METHOD Completing : BOOL
VAR_INPUT
    SequenceState : REFERENCE TO UDINT;
END_VAR
Completing := TRUE;
END_METHOD

METHOD Execute : BOOL
VAR_INPUT
    SequenceState : REFERENCE TO UDINT;
END_VAR
Execute := TRUE;
END_METHOD

METHOD Held : BOOL
VAR_INPUT
    SequenceState : REFERENCE TO UDINT;
END_VAR
Held := TRUE;
END_METHOD

METHOD Holding : BOOL
VAR_INPUT
    SequenceState : REFERENCE TO UDINT;
END_VAR
Holding := TRUE;
END_METHOD

METHOD Idle : BOOL
VAR_INPUT
    SequenceState : REFERENCE TO UDINT;
END_VAR
Idle := TRUE;
END_METHOD

METHOD Resetting : BOOL
VAR_INPUT
    SequenceState : REFERENCE TO UDINT;
END_VAR
Resetting := TRUE;
END_METHOD

METHOD Starting : BOOL
VAR_INPUT
    SequenceState : REFERENCE TO UDINT;
END_VAR
Starting := TRUE;
END_METHOD

METHOD Stopped : BOOL
VAR_INPUT
    SequenceState : REFERENCE TO UDINT;
END_VAR
Stopped := TRUE;
END_METHOD

METHOD Stopping : BOOL
VAR_INPUT
    SequenceState : REFERENCE TO UDINT;
END_VAR
Stopping := TRUE;
END_METHOD

METHOD Suspended : BOOL
VAR_INPUT
    SequenceState : REFERENCE TO UDINT;
END_VAR
Suspended := TRUE;
END_METHOD

METHOD Suspending : BOOL
VAR_INPUT
    SequenceState : REFERENCE TO UDINT;
END_VAR
Suspending := TRUE;
END_METHOD

METHOD Unholding : BOOL
VAR_INPUT
    SequenceState : REFERENCE TO UDINT;
END_VAR
Unholding := TRUE;
END_METHOD

METHOD Unsuspending : BOOL
VAR_INPUT
    SequenceState : REFERENCE TO UDINT;
END_VAR
Unsuspending := TRUE;
END_METHOD

(* This Module will be done initialize when ModuleInitialized := TRUE;, subequently all subitems will be called to be initialized *)
METHOD Initializing
END_METHOD

METHOD OnCyclicCall
END_METHOD

PROPERTY Statemachine : I_Statemachine
GET
Statemachine := _Statemachine;
END_GET
END_PROPERTY

END_FUNCTION_BLOCK

// Statemachine/PackML/PackMLStatemachine
FUNCTION_BLOCK PackMLStatemachine EXTENDS CyclicComponent IMPLEMENTS I_StateMachine
VAR
	StateList	   : StateList<17>;
	StateMachine   : FB_PMLStateMachine;
	StateCommand   : E_PMLCommand;
	_CurrentState  : E_PMLState;
	ModeController : PackMLModeControl := (StateMachine := THIS^);
END_VAR

PROPERTY Mode : I_Mode
GET
Mode := ModeController;
END_GET
SET
// Fix defined in PackML
END_SET
END_PROPERTY

METHOD PROTECTED CallState : BOOL
VAR_INPUT
	StateIndex : E_PMLState;
END_VAR

VAR
	State : I_State;
	i	  : DINT;
END_VAR
State := StateList.GetStateAtIndex(StateIndex);
IF State <> 0 THEN
	CallState := State.Executing();
ELSE
	CallState := TRUE;
END_IF

FOR i := 0 TO StateList.NumberOfStates DO
	State := StateList.GetStateAtIndex(i);
	IF State <> 0 AND i <> StateIndex THEN
		State.Inactive();
	END_IF
END_FOR
END_METHOD

METHOD ChangeState
VAR_INPUT
	StateCommand : DINT;
END_VAR
IF StateCommand <= 0 OR StateCommand > 17 THEN
	Trace.LogMessage('PackML Statemachine ChangeState()', 'StateId is not a PackML State');
END_IF

{warning disable C0196}
THIS^.StateCommand := StateCommand;
END_METHOD

{attribute 'monitoring' := 'call'}
PROPERTY CurrentState : DINT
GET
CurrentState := _CurrentState;
END_GET
END_PROPERTY

PROPERTY States : I_StateList
GET
States := StateList;
END_GET
END_PROPERTY

METHOD CyclicLogic
VAR_INST
	ClearingTon : TON;
END_VAR
IF StateList.NumberOfStates = 0 THEN
	RETURN;
END_IF

ModeController.CyclicLogic();
IF _CurrentState = E_PMLState.Undefined AND Mode.CurrentMode <> 0 THEN
	StateCommand := E_PMLCommand.Abort;
END_IF

StateMachine(eMode			  := TO_DINT(Mode.CurrentMode),
			 eCommand		  := StateCommand,
			 stSubUnitInfoRef :=,
			 stOptions		  :=,
			 eState			  => _CurrentState,
			 sState			  =>,
			 bError			  =>,
			 nErrorID		  =>);

CASE _CurrentState OF
	E_PMLState.Undefined:
		CallState(_CurrentState);

	E_PMLState.Clearing:
		ClearingTon(IN := TRUE, PT := CoreParameter.ClearingTimeout);
		IF CallState(_CurrentState) THEN
			ClearingTon(IN := FALSE);
			StateMachine.M_StateComplete();
		END_IF

		IF ClearingTon.Q THEN
			ClearingTon(IN := FALSE);
			Trace.LogMessage('Clearing Timeout exeeded!', 'CoreParameter.ClearingTimeout');
			StateCommand := E_PMLCommand.Abort;
		END_IF

	E_PMLState.Stopped:
		CallState(_CurrentState);

	E_PMLState.Starting:
		IF CallState(_CurrentState) THEN
			StateMachine.M_StateComplete();
		END_IF

	E_PMLState.Idle:
		CallState(_CurrentState);

	E_PMLState.Suspended:
		CallState(_CurrentState);

	E_PMLState.Execute:
		CallState(_CurrentState);

	E_PMLState.Stopping:
		IF CallState(_CurrentState) THEN
			StateMachine.M_StateComplete();
		END_IF

	E_PMLState.Aborting:
		IF CallState(_CurrentState) THEN
			StateMachine.M_StateComplete();
		END_IF

	E_PMLState.Aborted:
		CallState(_CurrentState);

	E_PMLState.Holding:
		IF CallState(_CurrentState) THEN
			StateMachine.M_StateComplete();
		END_IF

	E_PMLState.Held:
		CallState(_CurrentState);

	E_PMLState.Unholding:
		IF CallState(_CurrentState) THEN
			StateMachine.M_StateComplete();
		END_IF

	E_PMLState.Suspending:
		IF CallState(_CurrentState) THEN
			StateMachine.M_StateComplete();
		END_IF

	E_PMLState.Unsuspending:
		IF CallState(_CurrentState) THEN
			StateMachine.M_StateComplete();
		END_IF

	E_PMLState.Resetting:
		IF CallState(_CurrentState) THEN
			StateMachine.M_StateComplete();
		END_IF

	E_PMLState.Completing:
		IF CallState(_CurrentState) THEN
			StateMachine.M_StateComplete();
		END_IF

	E_PMLState.Completed:
		CallState(_CurrentState);
END_CASE
END_METHOD

END_FUNCTION_BLOCK

// Project Information/F_GetCompany
// This function has been automatically generated from the project information.
{attribute 'signature_flag' := '1073741824'}
{attribute 'TcGenerated'}
{attribute 'no-analysis'}
FUNCTION F_GetCompany : WSTRING
VAR_INPUT
	
END_VAR

F_GetCompany := "Beckhoff Automation LLC";

END_FUNCTION

// Project Information/F_GetTitle
// This function has been automatically generated from the project information.
{attribute 'signature_flag' := '1073741824'}
{attribute 'TcGenerated'}
{attribute 'no-analysis'}
FUNCTION F_GetTitle : WSTRING
VAR_INPUT
	
END_VAR

F_GetTitle := "Core";

END_FUNCTION

// Project Information/F_GetVersion
// This function has been automatically generated from the project information.
{attribute 'signature_flag' := '1073741824'}
{attribute 'TcGenerated'}
{attribute 'no-analysis'}
FUNCTION F_GetVersion : ST_LibVersion
VAR_INPUT
	
END_VAR

F_GetVersion.iMajor := 1;
F_GetVersion.iMinor := 2;
F_GetVersion.iBuild := 0;
F_GetVersion.iRevision := 0;
F_GetVersion.sVersion := '1.2.0';
F_GetVersion.nFlags := 0;

END_FUNCTION

// Statemachine/Generic/NextMinorStep
FUNCTION NextMinorStep : UDINT
VAR_IN_OUT
	StateVar : UDINT;
END_VAR

NextMinorStep := StateVar := StateVar + 1;

END_FUNCTION

// Statemachine/Generic/NextStep
FUNCTION NextStep : UDINT
VAR_IN_OUT
	StateVar : UDINT;
END_VAR

NextStep := StateVar := ((StateVar / 10) * 10) + 10;

END_FUNCTION

// Statemachine/Generic/Statemachine_HMI
FUNCTION_BLOCK Statemachine_HMI EXTENDS HmiFunction
VAR
	Statemachine : I_Statemachine;
	{ attribute 'TcHmiSymbol.AddSymbol' }
	{ attribute 'TcHmiSymbol.AddSymbol.UserGroups' := '__SystemAdministrators,Admin' }
	Statemachine_HMI : ST_Statemachine_HMI;
END_VAR

METHOD CyclicLogic
VAR_INST
	LastModeChangeCommand  : DINT;
	LastStateChangeCommand : DINT;
END_VAR
Statemachine_HMI.Name		  := Statemachine.Name;
Statemachine_HMI.CurrentState := Statemachine.CurrentState;
Statemachine_HMI.CurrentMode  := Statemachine.Mode.CurrentMode;
Statemachine_HMI.HmiEnabled	  := Enabled;
IF Enabled THEN
	IF Statemachine_HMI.ModeChangeCommand <> 0 THEN
		Statemachine.Mode.ChangeMode(Statemachine_HMI.ModeChangeCommand);
		LastModeChangeCommand			   := Statemachine_HMI.ModeChangeCommand;
		Statemachine_HMI.ModeChangeCommand := 0;
	END_IF

	{warning disable C0196}
	IF Statemachine_HMI.StateChangeCommand <> 0 THEN
		Statemachine.ChangeState(TO_UDINT(Statemachine_HMI.StateChangeCommand));
		{warning disable C0195}
		LastStateChangeCommand				:= Statemachine_HMI.StateChangeCommand;
		Statemachine_HMI.StateChangeCommand := 0;
	END_IF
ELSE
	Statemachine_HMI.StateChangeCommand := 0;
	Statemachine_HMI.ModeChangeCommand	:= 0;
END_IF
END_METHOD

(*FB_Init is always available implicitly and it is used primarily for initialization.
The return value is not evaluated. For a specific influence, you can also declare the
methods explicitly and provide additional code there with the standard initialization
code. You can evaluate the return value.*)
METHOD FB_Init : BOOL
VAR_INPUT
	(* TRUE: the retain variables are initialized (reset warm / reset cold)*)
	bInitRetains : BOOL;

	(* TRUE: the instance will be copied to the copy code afterward (online change)   *)
	bInCopyCode	 : BOOL;
	Name		 : T_MaxString;
	Statemachine : I_Statemachine;
END_VAR
THIS^.Statemachine := Statemachine;
ControlType		   := 'Statemachine';
LinkObject		   := 'Statemachine_HMI';
END_METHOD

END_FUNCTION_BLOCK

// Statemachine/PackML/NextAvailablePackMLCommands
FUNCTION_BLOCK NextAvailablePackMLCommands
VAR
	NextAvailableCommands : ARRAY[0..MAX_AVAILABLE_COMMANDS] OF E_PMLCommand;
	i					  : UDINT;
END_VAR

VAR CONSTANT
	MAX_AVAILABLE_COMMANDS : UDINT := 9;
END_VAR

METHOD PUBLIC GetCommands : ARRAY[0..MAX_AVAILABLE_COMMANDS] OF E_PMLCommand
VAR_INPUT
	CurrentMode	 : DINT(0..31);
	CurrentState : E_PMLState;
END_VAR

VAR
	ModeConfiguration : Tc3_PackML_V3.ST_PMLUnitModeConfiguration;
END_VAR
FOR i := 1 TO MAX_AVAILABLE_COMMANDS DO
	NextAvailableCommands[i] := E_PMLCommand.Undefined;
END_FOR

i				  := 0;
ModeConfiguration := Tc3_PackML_V3.GlobalVariables.stPMLUnitModeConfiguration[CurrentMode];
// Generate next possible Commands
CASE CurrentState OF
	E_PMLState.Undefined:
		;

	E_PMLState.Aborting:
		;

	E_PMLState.Aborted:
		NextAvailableCommands[i] := E_PMLCommand.Clear;

	E_PMLState.Clearing:
		;

	E_PMLState.Stopping:
		NextAvailableCommands[i] := E_PMLCommand.Abort;

	E_PMLState.Stopped:
		NextAvailableCommands[i] := E_PMLCommand.Abort;
		i						 := i + 1;
		IF NOT ModeConfiguration.aStateDisabled[E_PMLState.Resetting] AND NOT ModeConfiguration.aStateDisabled[E_PMLState.Idle] THEN
			NextAvailableCommands[i] := E_PMLCommand.Reset;
		ELSE
			NextAvailableCommands[i] := E_PMLCommand.Start;
		END_IF

	E_PMLState.Resetting:
		NextAvailableCommands[i] := E_PMLCommand.Abort;
		i						 := i + 1;
		NextAvailableCommands[i] := E_PMLCommand.Stop;

	E_PMLState.Idle:
		NextAvailableCommands[i] := E_PMLCommand.Abort;
		i						 := i + 1;
		NextAvailableCommands[i] := E_PMLCommand.Stop;
		i						 := i + 1;
		NextAvailableCommands[i] := E_PMLCommand.Start;

	E_PMLState.Starting:
		NextAvailableCommands[i] := E_PMLCommand.Abort;
		i						 := i + 1;
		NextAvailableCommands[i] := E_PMLCommand.Stop;

	E_PMLState.Execute:
		NextAvailableCommands[i] := E_PMLCommand.Abort;
		i						 := i + 1;
		NextAvailableCommands[i] := E_PMLCommand.Stop;
		i						 := i + 1;
		IF (NOT ModeConfiguration.aStateDisabled[E_PMLState.Held] AND NOT ModeConfiguration.aStateDisabled[E_PMLState.Holding]) OR (NOT ModeConfiguration.aStateDisabled[E_PMLState.Held] AND NOT ModeConfiguration.aStateDisabled[E_PMLState.Unholding]) THEN
			NextAvailableCommands[i] := E_PMLCommand.Hold;
			i						 := i + 1;
		END_IF

		IF (NOT ModeConfiguration.aStateDisabled[E_PMLState.Suspended] AND NOT ModeConfiguration.aStateDisabled[E_PMLState.Suspending]) OR (NOT ModeConfiguration.aStateDisabled[E_PMLState.Suspended] AND NOT ModeConfiguration.aStateDisabled[E_PMLState.Unsuspending]) THEN
			NextAvailableCommands[i] := E_PMLCommand.Suspend;
			i						 := i + 1;
		END_IF

		IF NOT ModeConfiguration.aStateDisabled[E_PMLState.Completed] AND NOT ModeConfiguration.aStateDisabled[E_PMLState.Completing] THEN
			NextAvailableCommands[i] := E_PMLCommand.Complete;
			i						 := i + 1;
		ELSIF NOT ModeConfiguration.aStateDisabled[E_PMLState.Resetting] THEN
			NextAvailableCommands[i] := E_PMLCommand.Reset;
			i						 := i + 1;
		END_IF

	E_PMLState.Completing:
		NextAvailableCommands[i] := E_PMLCommand.Abort;
		i						 := i + 1;
		NextAvailableCommands[i] := E_PMLCommand.Stop;

	E_PMLState.Completed:
		NextAvailableCommands[i] := E_PMLCommand.Abort;
		i						 := i + 1;
		NextAvailableCommands[i] := E_PMLCommand.Stop;
		i						 := i + 1;
		IF NOT ModeConfiguration.aStateDisabled[E_PMLState.Resetting] AND NOT ModeConfiguration.aStateDisabled[E_PMLState.Idle] THEN
			NextAvailableCommands[i] := E_PMLCommand.Reset;
		ELSE
			NextAvailableCommands[i] := E_PMLCommand.Start;
		END_IF

	E_PMLState.Holding:
		NextAvailableCommands[i] := E_PMLCommand.Abort;
		i						 := i + 1;
		NextAvailableCommands[i] := E_PMLCommand.Stop;

	E_PMLState.Held:
		NextAvailableCommands[i] := E_PMLCommand.Abort;
		i						 := i + 1;
		NextAvailableCommands[i] := E_PMLCommand.Stop;
		i						 := i + 1;
		NextAvailableCommands[i] := E_PMLCommand.Unhold;

	E_PMLState.Unholding:
		NextAvailableCommands[i] := E_PMLCommand.Abort;
		i						 := i + 1;
		NextAvailableCommands[i] := E_PMLCommand.Stop;

	E_PMLState.Suspending:
		NextAvailableCommands[i] := E_PMLCommand.Abort;
		i						 := i + 1;
		NextAvailableCommands[i] := E_PMLCommand.Stop;

	E_PMLState.Suspended:
		NextAvailableCommands[i] := E_PMLCommand.Abort;
		i						 := i + 1;
		NextAvailableCommands[i] := E_PMLCommand.Stop;
		i						 := i + 1;
		NextAvailableCommands[i] := E_PMLCommand.Unsuspend;

	E_PMLState.Unsuspending:
		NextAvailableCommands[i] := E_PMLCommand.Abort;
		i						 := i + 1;
		NextAvailableCommands[i] := E_PMLCommand.Stop;
END_CASE

GetCommands := NextAvailableCommands;
END_METHOD

END_FUNCTION_BLOCK

// Statemachine/PackML/PackMLStatemachine_HMI
FUNCTION_BLOCK PackMLStatemachine_HMI EXTENDS HmiFunction
VAR
	Statemachine				: I_Statemachine;
	NextAvailablePackMLCommands : NextAvailablePackMLCommands;
	{ attribute 'TcHmiSymbol.AddSymbol' }
	{ attribute 'TcHmiSymbol.AddSymbol.UserGroups' := '__SystemAdministrators,Admin' }
	Statemachine_HMI : ST_PackMLStatemachine_HMI;
END_VAR

METHOD CyclicLogic
VAR_INST
	LastModeChangeCommand  : DINT;
	LastStateChangeCommand : UDINT;
END_VAR
{warning disable C0196}
Statemachine_HMI.CurrentState := Statemachine.CurrentState;
Statemachine_HMI.CurrentMode  := Statemachine.Mode.CurrentMode;
Statemachine_HMI.Name		  := Statemachine.Name;
Statemachine_HMI.HmiEnabled	  := Enabled;
IF Enabled THEN
	IF Statemachine_HMI.ModeCommand <> 0 THEN
		Statemachine.Mode.ChangeMode(Statemachine_HMI.ModeCommand);
		LastModeChangeCommand		 := Statemachine_HMI.ModeCommand;
		Statemachine_HMI.ModeCommand := 0;
	END_IF

	{warning disable C0196}
	IF Statemachine_HMI.StateCommand <> 0 THEN
		Statemachine.ChangeState(TO_UDINT(Statemachine_HMI.StateCommand));
		{warning disable C0195}
		LastStateChangeCommand		  := Statemachine_HMI.StateCommand;
		Statemachine_HMI.StateCommand := 0;
	END_IF
ELSE
	Statemachine_HMI.StateCommand := 0;
	Statemachine_HMI.ModeCommand  := 0;
END_IF

Statemachine_HMI.NextAvailableCommands := NextAvailablePackMLCommands.GetCommands(Statemachine_HMI.CurrentMode, Statemachine_HMI.CurrentState);
END_METHOD

(*FB_Init is always available implicitly and it is used primarily for initialization.
The return value is not evaluated. For a specific influence, you can also declare the
methods explicitly and provide additional code there with the standard initialization
code. You can evaluate the return value.*)
METHOD FB_Init : BOOL
VAR_INPUT
	(* TRUE: the retain variables are initialized (reset warm / reset cold)*)
	bInitRetains : BOOL;

	(* TRUE: the instance will be copied to the copy code afterward (online change)   *)
	bInCopyCode	 : BOOL;
	Name		 : T_MaxString;
	Statemachine : I_Statemachine;
END_VAR
THIS^.Statemachine := Statemachine;
ControlType		   := 'PackMLStatemachine';
LinkObject		   := 'Statemachine_HMI';
END_METHOD

END_FUNCTION_BLOCK

// Visitors/Enable/CheckComponentsEnabledVisitor
FUNCTION_BLOCK CheckComponentsEnabledVisitor IMPLEMENTS I_ComponentVisitor
VAR
	Enablable : I_Enablable;
	_Enabled  : BOOL;
END_VAR

METHOD Check
VAR_INPUT
	Components : I_ComponentCollection;
END_VAR
_Enabled := TRUE;
Components.Accept(THIS^);
END_METHOD

{attribute 'monitoring' := 'call'}
PROPERTY Enabled : BOOL
GET
Enabled := _Enabled;
END_GET
END_PROPERTY

METHOD VisitComponent
VAR_INPUT
	Component : I_Component;
END_VAR
IF __QUERYINTERFACE(Component, Enablable) THEN
	IF NOT Enablable.Enabled THEN
		_Enabled := FALSE;
	END_IF
END_IF
END_METHOD

END_FUNCTION_BLOCK

// Visitors/Enable/DisableAllComponentsVisitor
FUNCTION_BLOCK DisableAllComponentsVisitor IMPLEMENTS I_ComponentVisitor
VAR
	Enablable : I_Enablable;
	_Enabled  : BOOL;
END_VAR

METHOD Disable
VAR_INPUT
	Components : I_ComponentCollection;
END_VAR
_Enabled := FALSE;
Components.Accept(THIS^);
END_METHOD

{attribute 'monitoring' := 'call'}
PROPERTY Enabled : BOOL
GET
Enabled := _Enabled;
END_GET
END_PROPERTY

METHOD VisitComponent
VAR_INPUT
	Component : I_Component;
END_VAR
IF __QUERYINTERFACE(Component, Enablable) THEN
	Enablable.Disable();
	IF Enablable.Enabled THEN
		_Enabled := TRUE;
	END_IF
END_IF
END_METHOD

END_FUNCTION_BLOCK

// Visitors/Enable/EnableAllComponentsVisitor
FUNCTION_BLOCK EnableAllComponentsVisitor IMPLEMENTS I_ComponentVisitor
VAR
	Enablable	   : I_Enablable;
	_Enabled	   : BOOL;
	ErrorComponent : I_Component;
END_VAR

METHOD Enable
VAR_INPUT
	Components : I_ComponentCollection;
END_VAR
_Enabled := TRUE;
Components.Accept(THIS^);
END_METHOD

{attribute 'monitoring' := 'call'}
PROPERTY Enabled : BOOL
GET
Enabled := _Enabled;
END_GET
END_PROPERTY

METHOD VisitComponent
VAR_INPUT
	Component : I_Component;
END_VAR
IF __QUERYINTERFACE(Component, Enablable) THEN
	Enablable.Enable();
	IF NOT Enablable.Enabled THEN
		ErrorComponent := Component;
		_Enabled	   := FALSE;
	END_IF
END_IF
END_METHOD

END_FUNCTION_BLOCK

// Visitors/Events/GetActiveEventSeverityVisitor
FUNCTION_BLOCK GetActiveEventSeverityVisitor IMPLEMENTS I_ModuleVisitor, I_ComponentVisitor
VAR
	EntryModule			 : I_Module;
	HighestEventSeverity : TcEventSeverity;
	TcEventClass		 : I_EventClassTcEvents;
END_VAR

PROPERTY ActiveEventSeverity : TcEventSeverity
GET
HighestEventSeverity := Global.TcEventSeverity.Verbose;
EntryModule.Accept(THIS^);
ActiveEventSeverity := HighestEventSeverity;
END_GET
END_PROPERTY

(*FB_Init is always available implicitly and it is used primarily for initialization.
The return value is not evaluated. For a specific influence, you can also declare the
methods explicitly and provide additional code there with the standard initialization
code. You can evaluate the return value.*)
METHOD FB_Init : BOOL
VAR_INPUT
	(* TRUE: the retain variables are initialized (reset warm / reset cold)*)
	bInitRetains : BOOL;

	(* TRUE: the instance will be copied to the copy code afterward (online change)   *)
	bInCopyCode : BOOL;
	EntryModule : I_Module;
END_VAR
THIS^.EntryModule := EntryModule;
END_METHOD

METHOD VisitComponent
VAR_INPUT
	Component : I_Component;
END_VAR

VAR
	Severity : TcEventSeverity;
END_VAR
IF __QUERYINTERFACE(Component, TcEventClass) THEN
	Severity := TcEventClass.GetHighestActiveEventSeverity();
	IF Severity > HighestEventSeverity THEN
		HighestEventSeverity := Severity;
	END_IF
END_IF
END_METHOD

METHOD VisitModule
VAR_INPUT
	Module : I_Module;
END_VAR

VAR
	Severity : TcEventSeverity;
END_VAR
Module.Components.Accept(THIS^);
Module.Modules.Accept(THIS^);
IF __QUERYINTERFACE(Module, TcEventClass) THEN
	Severity := TcEventClass.GetHighestActiveEventSeverity();
	IF Severity > HighestEventSeverity THEN
		HighestEventSeverity := Severity;
	END_IF
END_IF
END_METHOD

END_FUNCTION_BLOCK

// Visitors/HMI/GetSystemTreeJsonHmiVisitor
FUNCTION_BLOCK GetSystemTreeJsonHmiVisitor
VAR_GENERIC CONSTANT
	TreeMax : UDINT := 10000;
END_VAR IMPLEMENTS I_ModuleVisitor, I_ComponentVisitor
VAR
	{ attribute 'TcHmiSymbol.AddSymbol' }
	{ attribute 'TcHmiSymbol.AddSymbol.UserGroups' := '__SystemAdministrators,Admin' }
	SystemHmiTree : STRING(TreeMax);
	{attribute 'hide'}
	Module : I_Module;
	{attribute 'hide'}
	HmiFunction : I_HmiFunction;
	{attribute 'hide'}
	Json : FB_JsonSaxWriter;
	{attribute 'hide'}
	Entry	 : T_MaxString;
	LinkRoot : STRING;
END_VAR

METHOD PRIVATE Clear
VAR_INPUT
END_VAR
MEMSET(ADR(SystemHmiTree), 0, SIZEOF(SystemHmiTree));
Json.ResetDocument();
END_METHOD

//FB_Init is always available implicitly and it is used primarily for initialization.

//The return value is not evaluated. For a specific influence, you can also declare the

//methods explicitly and provide additional code there with the standard initialization

//code. You can evaluate the return value.
METHOD FB_Init : BOOL
VAR_INPUT
	bInitRetains : BOOL; // TRUE: the retain variables are initialized (reset warm / reset cold)
	bInCopyCode	 : BOOL; // TRUE: the instance will be copied to the copy code afterward (online change)   
	LinkRoot	 : STRING;
END_VAR
THIS^.LinkRoot := LinkRoot;
END_METHOD

METHOD GetTree
VAR_INPUT
	EntryModule : I_Module;
END_VAR
IF EntryModule = 0 THEN
	RETURN;
END_IF

Module := EntryModule;
Clear();
Json.StartObject();
Entry := Module.Name;
Json.AddKey(Entry);
Json.StartArray();
Module.Components.Accept(THIS^);
Json.EndArray();
Module.Modules.Accept(THIS^);
Json.EndObject();
Json.CopyDocument(pDoc := SystemHmiTree, nDoc := SIZEOF(SystemHmiTree));
END_METHOD

METHOD VisitComponent
VAR_INPUT
	Component : I_Component;
END_VAR
IF __QUERYINTERFACE(Component, HmiFunction) THEN
	Json.StartObject();
	Entry := HmiFunction.ControlType;
	Json.AddKeyString('ControlType', Entry);
	Entry := RIGHT(HmiFunction.InstancePath, (LEN(HmiFunction.InstancePath) - FIND(HmiFunction.InstancePath, LinkRoot)) + 1);
	Entry := CONCAT(CONCAT(Entry, '.'), HmiFunction.LinkObject);
	Json.AddKeyString('LinkPath', Entry);
	Json.EndObject();
END_IF
END_METHOD

METHOD VisitModule
VAR_INPUT
	Module : I_Module;
END_VAR
Entry := Module.Name;
IF Entry <> '' THEN
	Json.AddKey(Entry);
	Json.StartArray();
	Module.Components.Accept(THIS^);
	Json.EndArray();
	Module.Modules.Accept(THIS^);
END_IF
END_METHOD

END_FUNCTION_BLOCK

// Visitors/HMI/HmiEnableDisableAllVisitor
FUNCTION_BLOCK HmiEnableDisableAllVisitor IMPLEMENTS I_ComponentVisitor, I_ModuleVisitor
VAR
	{attribute 'hide'}
	HmiFunction : I_HmiFunction;
	{attribute 'hide'}
	Enable : BOOL;
END_VAR

METHOD DisableHmi
VAR_INPUT
	Module : I_Module;
END_VAR
Enable := FALSE;
Module.Accept(THIS^);
END_METHOD

METHOD EnableHmi
VAR_INPUT
	Module : I_Module;
END_VAR
Enable := TRUE;
Module.Accept(THIS^);
END_METHOD

METHOD VisitComponent
VAR_INPUT
	Component : I_Component;
END_VAR
IF __QUERYINTERFACE(Component, HmiFunction) THEN
	IF Enable THEN
		HmiFunction.Enable();
	ELSE
		HmiFunction.Disable();
	END_IF
END_IF
END_METHOD

METHOD VisitModule
VAR_INPUT
	Module : I_Module;
END_VAR
Module.Components.Accept(THIS^);
Module.Modules.Accept(THIS^);
END_METHOD

END_FUNCTION_BLOCK

// Visitors/Override/SetAllOverrideVisitor
FUNCTION_BLOCK SetAllOverrideVisitor IMPLEMENTS I_ModuleVisitor, I_ComponentVisitor
VAR
	ipOverride : I_Override;
	_Override  : LREAL;
END_VAR

METHOD Set
VAR_INPUT
	Module	 : I_Module;
	Override : LREAL;
END_VAR
_Override := Override;
Module.Accept(THIS^);
IF __QUERYINTERFACE(Module, ipOverride) THEN
	ipOverride.Override := _Override;
END_IF
END_METHOD

METHOD VisitComponent
VAR_INPUT
	Component : I_Component;
END_VAR
IF __QUERYINTERFACE(Component, ipOverride) THEN
	ipOverride.Override := _Override;
END_IF
END_METHOD

METHOD VisitModule
VAR_INPUT
	Module : I_Module;
END_VAR
Module.Components.Accept(THIS^);
Module.Modules.Accept(THIS^);
IF __QUERYINTERFACE(Module, ipOverride) THEN
	ipOverride.Override := _Override;
END_IF
END_METHOD

END_FUNCTION_BLOCK

// Visitors/PackML Statemachine/ChangePackMLStateOnAllSubModulesVisitor
FUNCTION_BLOCK ChangePackMLStateOnAllSubModulesVisitor IMPLEMENTS I_ModuleVisitor
VAR
	PackMLCommand : E_PMLCommand;
	Statemachine  : I_ContainStatemachine;
	StateChanged  : BOOL;
	CheckState	  : E_PMLState;
END_VAR

METHOD ChangeState : BOOL;
VAR_INPUT
	PackMLCommand : E_PMLCommand;
	Module		  : I_Module;
END_VAR
StateChanged		:= TRUE;
THIS^.PackMLCommand := PackMLCommand;
CASE THIS^.PackMLCommand OF
	E_PMLCommand.Abort:
		CheckState := E_PMLState.Aborted;

	E_PMLCommand.Clear, E_PMLCommand.Stop:
		CheckState := E_PMLState.Stopped;

	E_PMLCommand.Complete:
		CheckState := E_PMLState.Completed;

	E_PMLCommand.Hold:
		CheckState := E_PMLState.Held;

	E_PMLCommand.Reset:
		CheckState := E_PMLState.Idle;

	E_PMLCommand.Start, E_PMLCommand.Unhold, E_PMLCommand.Unsuspend:
		CheckState := E_PMLState.Execute;

	E_PMLCommand.Suspend:
		CheckState := E_PMLState.Suspended;

	E_PMLCommand.Undefined:
		CheckState := E_PMLState.Undefined;
END_CASE

Module.Modules.Accept(THIS^);
ChangeState := StateChanged;
END_METHOD

METHOD VisitModule
VAR_INPUT
	Module : I_Module;
END_VAR

VAR_INST
	ReturnModule : I_Module;
END_VAR
IF __QUERYINTERFACE(Module, Statemachine) THEN
	IF Statemachine.Statemachine = 0 THEN
		ReturnModule := Module;
		RETURN;
	END_IF

	Statemachine.Statemachine.ChangeState(THIS^.PackMLCommand);
	IF Statemachine.Statemachine.CurrentState <> CheckState THEN
		StateChanged := FALSE;
	END_IF
END_IF
END_METHOD

END_FUNCTION_BLOCK

// Visitors/PackML Statemachine/EventReactorPackMLVisitor
FUNCTION_BLOCK EventReactorPackMLVisitor EXTENDS CyclicComponent IMPLEMENTS I_ModuleVisitor, I_ComponentVisitor
VAR
	EntryModule			 : I_Module;
	HighestEventReaction : DINT;
	EventReaction		 : I_EventReaction;
	ModuleStatemachine	 : I_ContainStatemachine;
	ReactedName			 : T_MaxString;
END_VAR

METHOD CyclicLogic
IF ModuleStatemachine = 0 THEN
	RETURN;
END_IF

HighestEventReaction := 0;
EntryModule.Accept(THIS^);
CASE HighestEventReaction OF
	0:	  // Verbose
	1:	  // Info
	2:	  // Warning
	3, 4: // Error & Critical
		IF ModuleStatemachine.Statemachine.CurrentState <> E_PMLState.Aborted AND ModuleStatemachine.Statemachine.CurrentState <> E_PMLState.Aborting AND ModuleStatemachine.Statemachine.CurrentState <> E_PMLState.Clearing THEN
			Trace.LogMessage('Module or Component leading to reaction', ReactedName);
			ModuleStatemachine.Statemachine.ChangeState(E_PMLCommand.Abort);
			ReactedName := '';
		END_IF
END_CASE
END_METHOD

(*FB_Init is always available implicitly and it is used primarily for initialization.
The return value is not evaluated. For a specific influence, you can also declare the
methods explicitly and provide additional code there with the standard initialization
code. You can evaluate the return value.*)
METHOD FB_Init : BOOL
VAR_INPUT
	(* TRUE: the retain variables are initialized (reset warm / reset cold)*)
	bInitRetains : BOOL;

	(* TRUE: the instance will be copied to the copy code afterward (online change)   *)
	bInCopyCode : BOOL;
	Name		: T_MaxString;
	EntryModule : I_Module;
END_VAR
THIS^.EntryModule := EntryModule;
__QUERYINTERFACE(EntryModule, ModuleStatemachine);
END_METHOD

METHOD VisitComponent
VAR_INPUT
	Component : I_Component;
END_VAR

VAR
	Reaction : DINT;
END_VAR
IF __QUERYINTERFACE(Component, EventReaction) THEN
	Reaction := EventReaction.GetHighestActiveEventReaction();
	IF Reaction > HighestEventReaction THEN
		IF ReactedName = '' THEN
			ReactedName := Component.Name;
		END_IF

		HighestEventReaction := Reaction;
	END_IF
END_IF
END_METHOD

METHOD VisitModule
VAR_INPUT
	Module : I_Module;
END_VAR

VAR
	Reaction : DINT;
END_VAR
Module.Components.Accept(THIS^);
Module.Modules.Accept(THIS^);
IF __QUERYINTERFACE(Module, EventReaction) THEN
	Reaction := EventReaction.GetHighestActiveEventReaction();
	IF Reaction > HighestEventReaction THEN
		IF ReactedName = '' THEN
			ReactedName := Module.Name;
		END_IF

		HighestEventReaction := Reaction;
	END_IF
END_IF
END_METHOD

END_FUNCTION_BLOCK

// Visitors/Reset/GetComponentsTaskResultVisitor
FUNCTION_BLOCK GetComponentsTaskResultVisitor IMPLEMENTS I_ComponentVisitor, I_TaskResult
VAR
	{attribute 'hide'}
	Result : I_TaskResult;
	{attribute 'hide'}
	_Busy : BOOL;
	{attribute 'hide'}
	_Error : BOOL;
	{attribute 'hide'}
	_ErrorId : UDINT;
END_VAR

{attribute 'monitoring' := 'call'}
PROPERTY Busy : BOOL
GET
Busy := _Busy;
END_GET
END_PROPERTY

{attribute 'monitoring' := 'call'}
PROPERTY Error : BOOL
GET
Error := _Error;
END_GET
END_PROPERTY

{attribute 'monitoring' := 'call'}
PROPERTY ErrorId : UDINT
GET
ErrorID := _ErrorID;
END_GET
END_PROPERTY

METHOD Update
VAR_INPUT
	Module : I_Module;
END_VAR
_Error	 := FALSE;
_ErrorId := 0;
_Busy	 := FALSE;
Module.Components.Accept(THIS^);
END_METHOD

METHOD VisitComponent
VAR_INPUT
	Component : I_Component;
END_VAR
IF __QUERYINTERFACE(Component, Result) THEN
	IF Result.Error THEN
		_Error	 := TRUE;
		_ErrorId := Result.ErrorId;
	END_IF

	IF Result.Busy THEN
		_Busy := TRUE;
	END_IF
END_IF
END_METHOD

END_FUNCTION_BLOCK

// Visitors/Reset/ResetAllVisitor
FUNCTION_BLOCK ResetAllVisitor IMPLEMENTS I_ModuleVisitor, I_ComponentVisitor, I_TaskResult
VAR
	{attribute 'hide'}
	Resettable : I_Resettable;
	{attribute 'hide'}
	Result : I_TaskResult;
	{attribute 'hide'}
	_Busy : BOOL;
	{attribute 'hide'}
	_Error : BOOL;
	{attribute 'hide'}
	_ErrorId	   : UDINT;
	ErrorComponent : I_Component;
	ErrorModule	   : I_Module;
END_VAR

{attribute 'monitoring' := 'call'}
PROPERTY Busy : BOOL
GET
Busy := _Busy;
END_GET
END_PROPERTY

{attribute 'monitoring' := 'call'}
PROPERTY Error : BOOL
GET
Error := _Error;
END_GET
END_PROPERTY

{attribute 'monitoring' := 'call'}
PROPERTY ErrorId : UDINT
GET
ErrorID := _ErrorID;
END_GET
END_PROPERTY

METHOD Reset
VAR_INPUT
	Module : I_Module;
END_VAR
_Error	 := FALSE;
_ErrorId := 0;
_Busy	 := FALSE;
Module.Accept(THIS^);
IF __QUERYINTERFACE(Module, Resettable) THEN
	Resettable.Reset();
END_IF

IF __QUERYINTERFACE(Module, Result) THEN
	IF Result.Error THEN
		_Error	 := TRUE;
		_ErrorId := Result.ErrorId;
	END_IF

	IF Result.Busy THEN
		_Busy := TRUE;
	END_IF
END_IF
END_METHOD

METHOD VisitComponent
VAR_INPUT
	Component : I_Component;
END_VAR
IF __QUERYINTERFACE(Component, Resettable) THEN
	Resettable.Reset();
END_IF

IF __QUERYINTERFACE(Component, Result) THEN
	IF Result.Error THEN
		ErrorComponent := Component;
		_Error		   := TRUE;
		_ErrorId	   := Result.ErrorId;
	END_IF

	IF Result.Busy THEN
		_Busy := TRUE;
	END_IF
END_IF
END_METHOD

METHOD VisitModule
VAR_INPUT
	Module : I_Module;
END_VAR
Module.Components.Accept(THIS^);
Module.Modules.Accept(THIS^);
IF __QUERYINTERFACE(Module, Resettable) THEN
	Resettable.Reset();
END_IF

IF __QUERYINTERFACE(Module, Result) THEN
	IF Result.Error THEN
		ErrorModule := Module;
		_Error		:= TRUE;
		_ErrorId	:= Result.ErrorId;
	END_IF

	IF Result.Busy THEN
		_Busy := TRUE;
	END_IF
END_IF
END_METHOD

END_FUNCTION_BLOCK

// Visitors/Statemachine/ChangeModeOnAllSubModulesVisitor
FUNCTION_BLOCK ChangeModeOnAllSubModulesVisitor IMPLEMENTS I_ModuleVisitor
VAR
	TargetMode	 : DINT;
	Statemachine : I_ContainStatemachine;
END_VAR

METHOD ChangeMode
VAR_INPUT
	TargetMode : DINT;
	Module	   : I_Module;
END_VAR
THIS^.TargetMode := TargetMode;
Module.Modules.Accept(THIS^);
END_METHOD

METHOD VisitModule
VAR_INPUT
	Module : I_Module;
END_VAR
IF __QUERYINTERFACE(Module, Statemachine) THEN
	Statemachine.Statemachine.Mode.ChangeMode(THIS^.TargetMode);
END_IF
END_METHOD

END_FUNCTION_BLOCK

// Visitors/Statemachine/ChangeStateOnAllSubModulesVisitor
FUNCTION_BLOCK ChangeStateOnAllSubModulesVisitor IMPLEMENTS I_ModuleVisitor
VAR
	TargetState	 : DINT;
	Statemachine : I_ContainStatemachine;
	StateChanged : BOOL;
END_VAR

METHOD ChangeState : BOOL
VAR_INPUT
	TargetState : DINT;
	Module		: I_Module;
END_VAR
StateChanged	  := TRUE;
THIS^.TargetState := TargetState;
Module.Modules.Accept(THIS^);
ChangeState := StateChanged;
END_METHOD

METHOD VisitModule
VAR_INPUT
	Module : I_Module;
END_VAR

VAR_INST
	ReturnModule : I_Module;
END_VAR
IF __QUERYINTERFACE(Module, Statemachine) THEN
	IF Statemachine.Statemachine = 0 THEN
		ReturnModule := Module;
		RETURN;
	END_IF

	Statemachine.Statemachine.ChangeState(THIS^.TargetState);
	IF Statemachine.Statemachine.CurrentState <> THIS^.TargetState THEN
		StateChanged := FALSE;
	END_IF
END_IF
END_METHOD

END_FUNCTION_BLOCK

// Visitors/Statemachine/EventReactorVisitor
FUNCTION_BLOCK EventReactorVisitor EXTENDS CyclicComponent IMPLEMENTS I_ModuleVisitor, I_ComponentVisitor
VAR
	EntryModule			 : I_Module;
	HighestEventReaction : DINT;
	EventReaction		 : I_EventReaction;
	ModuleStatemachine	 : I_ContainStatemachine;
END_VAR

METHOD CyclicLogic
IF ModuleStatemachine = 0 THEN
	RETURN;
END_IF

HighestEventReaction := 0;
EntryModule.Accept(THIS^);
CASE HighestEventReaction OF
	0: // Verbose
	1: // Info
	2: // Warning
	3: // Error
	4: // Critical
END_CASE
END_METHOD

(*FB_Init is always available implicitly and it is used primarily for initialization.
The return value is not evaluated. For a specific influence, you can also declare the
methods explicitly and provide additional code there with the standard initialization
code. You can evaluate the return value.*)
METHOD FB_Init : BOOL
VAR_INPUT
	(* TRUE: the retain variables are initialized (reset warm / reset cold)*)
	bInitRetains : BOOL;

	(* TRUE: the instance will be copied to the copy code afterward (online change)   *)
	bInCopyCode : BOOL;
	Name		: T_MaxString;
	EntryModule : I_Module;
END_VAR
THIS^.EntryModule := EntryModule;
__QUERYINTERFACE(EntryModule, ModuleStatemachine);
END_METHOD

METHOD VisitComponent
VAR_INPUT
	Component : I_Component;
END_VAR

VAR
	Reaction : DINT;
END_VAR
IF __QUERYINTERFACE(Component, EventReaction) THEN
	Reaction := EventReaction.GetHighestActiveEventReaction();
	IF Reaction > HighestEventReaction THEN
		HighestEventReaction := Reaction;
	END_IF
END_IF
END_METHOD

METHOD VisitModule
VAR_INPUT
	Module : I_Module;
END_VAR

VAR
	Reaction : DINT;
END_VAR
Module.Components.Accept(THIS^);
Module.Modules.Accept(THIS^);
IF __QUERYINTERFACE(Module, EventReaction) THEN
	Reaction := EventReaction.GetHighestActiveEventReaction();
	IF Reaction > HighestEventReaction THEN
		HighestEventReaction := Reaction;
	END_IF
END_IF
END_METHOD

END_FUNCTION_BLOCK

// Visitors/Stop/StopAllComponentsVisitor
FUNCTION_BLOCK StopAllComponentsVisitor IMPLEMENTS I_ComponentVisitor
VAR
	Stoppable : I_Stoppable;
	_Stopped  : BOOL;
END_VAR

METHOD Stop
VAR_INPUT
	Components : I_ComponentCollection;
END_VAR
_Stopped := TRUE;
Components.Accept(THIS^);
END_METHOD

{attribute 'monitoring' := 'call'}
PROPERTY Stopped : BOOL
GET
Stopped := _Stopped;
END_GET
END_PROPERTY

METHOD VisitComponent
VAR_INPUT
	Component : I_Component;
END_VAR
IF __QUERYINTERFACE(Component, Stoppable) THEN
	Stoppable.Stop();
	IF NOT Stoppable.Stopped THEN
		_Stopped := FALSE;
	END_IF
END_IF
END_METHOD

END_FUNCTION_BLOCK
